TYPE E_TcMatSimDataAreaType :
(
	NotSpecified := 0,
	Standard,
	InputSrc,
	InputDst,
	OutputSrc,
	OutputDst,
	InternalDa,
	MArea,
	RetainDa
);
END_TYPE

(* stored: Version 1.1.0.1, ProductVersion 3.1.4020.12
   DUT E_TcMatSimDataAreaType: Id {07b40632-877c-4a79-9984-71124dd39691} *)
